FUNCTION_BLOCK FB_StoneFurnace IMPLEMENTS I_2InputConversion
VAR
	iStoredrawproduct 			: UINT ; // Hoevelheid Erts in machine
	iStoredfuel			: UINT ; // Hoeveelheid kolen in machine
	iStoredProducts		: UINT ; // Aantal producten in voorraad
	tProductionTime		: TIME := T#3.3S; 
	tonProductionPulse 	: TON  ; // productie tick

	iMaxProducts		: UINT := 100 ; // maximum amount of stored products 
END_VAR

// run production timer
tonProductionPulse(pt := tProductionTime , IN := NOT tonProductionPulse.Q);

// produce product 
IF tonProductionPulse.Q THEN 
	Convert();
END_IF

METHOD PRIVATE Convert : BOOL
VAR_INPUT

END_VAR
VAR

END_VAR
// controleer of er Erts en kolen aanwezig zijn
IF iStoredrawproduct > 0 AND iStoredfuel > 0 AND iStoredProducts < iMaxProducts THEN 
	iStoredrawproduct 		:= iStoredrawproduct 		- 1;
	iStoredfuel		:= iStoredfuel		- 1;
	iStoredProducts	:= iStoredProducts	+ 1;
END_IF
END_METHOD

METHOD Input_1 : UINT
VAR_INPUT
	Amount : UINT ; // coal infeed amount 
END_VAR
VAR
	xTotal : UINT ; // internal total value	
END_VAR
xTotal := iStoredfuel + Amount;
IF xTotal <= iMaxProducts THEN 
	iStoredfuel := iStoredfuel + Amount;
	Input_1 := 0 ;
ELSE 
	Input_1 := Amount - iStoredfuel;
	iStoredfuel := iMaxProducts;
END_IF
END_METHOD

METHOD PUBLIC Input_2 : UINT
VAR_INPUT
	Amount : UINT ; // coal infeed amount 
END_VAR
VAR
	xTotal : UINT ; // internal total value	
END_VAR
xTotal := iStoredrawproduct + Amount;
IF xTotal <= iMaxProducts THEN 
	iStoredrawproduct := iStoredrawproduct + Amount;
	Input_2 := 0 ;
ELSE 
	Input_2 := Amount - iStoredrawproduct;
	iStoredrawproduct := iMaxProducts;
END_IF
END_METHOD

PROPERTY ProductsOut : UINT
GET
ProductsOut := iStoredProducts;
iStoredProducts := 0;
END_GET
END_PROPERTY

END_FUNCTION_BLOCK

(* stored: Version 1.1.0.1, ProductVersion 3.1.4024.13
   POU FB_StoneFurnace: Id {2f6fbf9f-40a3-40f7-af15-5a237660f659}, SpecialFunc None
   Method Convert: Id {f2d2bd65-dcf8-4fc1-813c-961dbd881ad5}
   Method Input_1: Id {baa7ed43-1775-4880-bff8-5323c1dbed6d}
   Method Input_2: Id {e49a2bd9-a430-4e5a-aa4f-08b2a8149d1f}
   Property ProductsOut: Id {4d9ff0ce-bf71-49c4-a607-e857d3f1c300}
   Get Get: Id {da49789d-4fb5-4d61-9302-43487c8b0c0b} *)
